		MYSQL_TYPE_BIT,
		MYSQL_TYPE_NEWDATE,
		MYSQL_TYPE_YEAR,
		MYSQL_TYPE_NULL,
		MYSQL_TYPE_ENUM,
		MYSQL_TYPE_SET,
		MYSQL_TYPE_TINY_BLOB,
		MYSQL_TYPE_MEDIUM_BLOB,
		MYSQL_TYPE_LONG_BLOB,
		MYSQL_TYPE_BLOB,
		MYSQL_TYPE_GEOMETRY : (* Unsupported MySQL-Data-Types *)
			sValue := CONCAT('CONVERT-ERROR: Unsupported MySQL-Data-Type: "', INT_TO_STRING(stQueryResult.astColumns[iCol-1].eType) );
			sValue := CONCAT(sValue, '"');
			MySql_GetStringValue := 16#80006008;
			;
	ELSE
		sValue := CONCAT('CONVERT-ERROR: Unknown MySQL-Data-Type: "', INT_TO_STRING(stQueryResult.astColumns[iCol-1].eType) );
		sValue := CONCAT(sValue, '"');
		MySql_GetStringValue := 16#80006007;
	END_CASE

END_IF

END_FUNCTION

// Device/Application/MYSQL/public/MySql_Version
FUNCTION MySql_Version : WORD
(*

 date     | release	| author  | Desc
----------+---------+------------------------------------------------------------
 21.03.14 |  3.8	| CM      | MySql_Query: New constant "gcMySql_tResponseCompliedlyReceived" 
 13.03.14 |  3.7	| CM      | MySql_Query: Initialisation of "stResultSet" now optional 
 02.07.12 |  3.6	| CM      | MySql_Query: BugFix for large SQL-Statements 
 17.04.12 |  3.5	| CM      | MySql_Query: BugFix for TIMEOUT error by "CALL <stored proc>"  
 25.01.12 |  3.4	| CM      | All: BugFix for large SQL statements 
 26.09.11 |  3.3	| CM      | MySql_Query: Clear complied result set before use 
 16.09.11 |  3.2	| CM      | MySql_Query: BugFix for large result sets 
 06.12.10 |  3.1    | CM      | MySql_GetStringValue: BugFix for Fieldtype 'TOD#'
 09.11.10 |  3.0    | CM      | MySql_Query: Optimize cycletime, "stResultSet" now VAR_IN_OUT prior VAR_OUTPUT  
 29.09.10 |  2.4    | CM      | MySql_Login: Bugfix for IP in dotted format
 28.09.10 |  2.3    | CM      | MySql_Login: Add DNS support for 750-881 and derivates
 28.09.10 |  2.2    | CM      | MySql_Login: Add error message when Login not allowed for this host
 19.08.10 |  2.1    | CM      | MySql_Query: ReceiveBuffer handling modified
 06.08.10 |  2.0	| CM      | Init - Switch from STRUCT "MySql" to FB "MySql_Context" 
 03.08.10 |  1.0	| CM      | Port to IEC 6-1131 
 22.06.09 |  0.0	| PEJ     | Original (C-Code)  
 
 *)
VAR_INPUT
END_VAR
VAR
	(* Current library version *)
	bMajor : BYTE := 16#03;
	bMinor : BYTE := 16#08;
END_VAR

MySql_Version := SHL(BYTE_TO_WORD(bMajor), 8) OR BYTE_TO_WORD(bMinor);

END_FUNCTION

// Device/Application/vis/Visualization
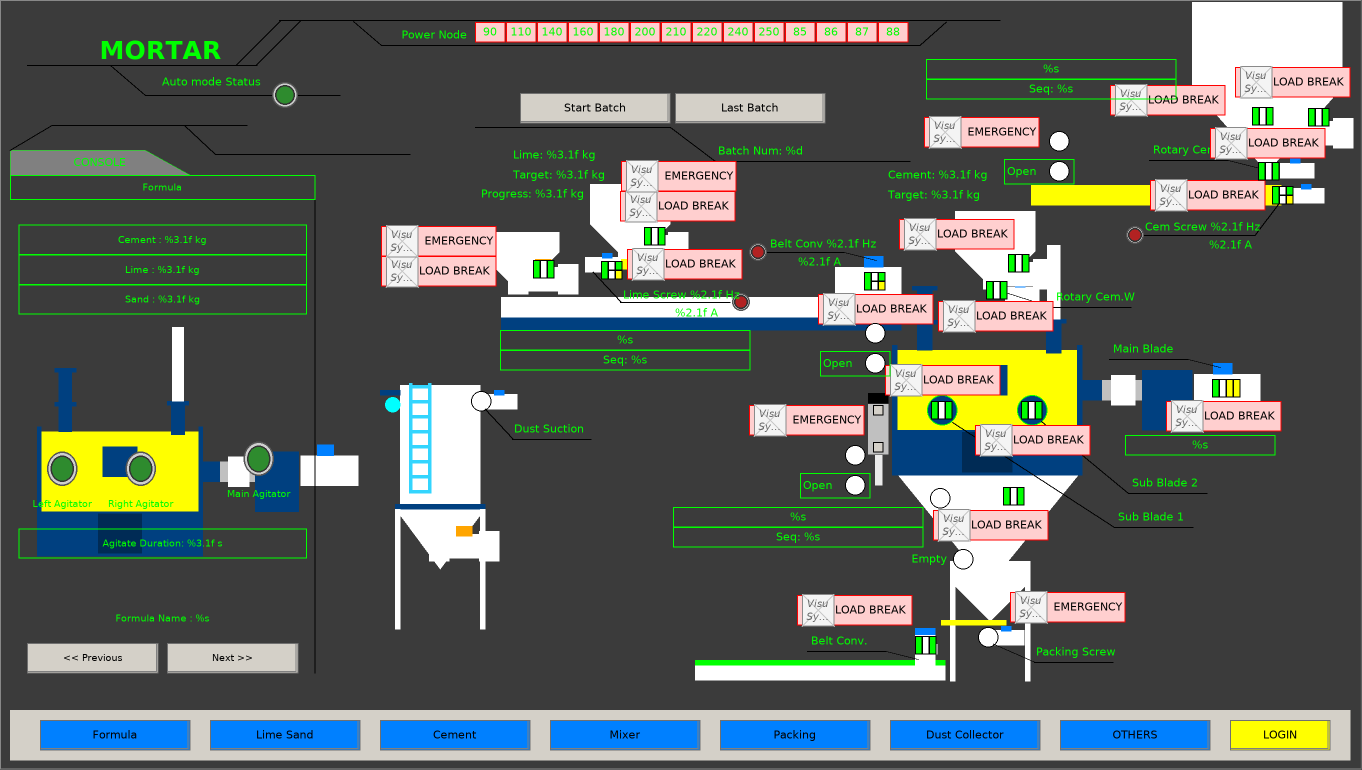
VISUALIZATION Visualization  // 1362x770
    Rectangle (800,473 70x25), "Open", colour toggle: DO381
    Rectangle (1004,159 70x25), "Open", colour toggle: DO371
    Line (1360,0) (1360,768)
    Rectangle (1031,185 250x20), angle 30
    Polygon (479,232) (559,232) (559,252) (519,292) (479,252)
    Rectangle (10,710 1340x50)
    Button (40,720 150x30), "Formula"
        OnMouseClick: FrameSelectionChange Selection=SelectedFrame=543ee2c1-9089-4e2a-a341-85b06829db8c, GlobSel=AssignType=Directly, SelType=Locally
    Button (210,720 150x30), "Lime Sand"
        OnMouseClick: FrameSelectionChange Selection=SelectedFrame=543ee2c1-9089-4e2a-a341-85b06829db8c, Selection=1, GlobSel=AssignType=Directly, SelType=Locally
    Button (380,720 150x30), "Cement"
        OnMouseClick: FrameSelectionChange Selection=SelectedFrame=543ee2c1-9089-4e2a-a341-85b06829db8c, Selection=2, GlobSel=AssignType=Directly, SelType=Locally
    Button (550,720 150x30), "Mixer"
        OnMouseClick: FrameSelectionChange Selection=SelectedFrame=543ee2c1-9089-4e2a-a341-85b06829db8c, Selection=3, GlobSel=AssignType=Directly, SelType=Locally
    Button (890,720 150x30), "Dust Collector"
        OnMouseClick: FrameSelectionChange Selection=SelectedFrame=543ee2c1-9089-4e2a-a341-85b06829db8c, Selection=4, GlobSel=AssignType=Directly, SelType=Locally
    Rectangle (1291,188 26x15), angle 30
    Rectangle (1301,184 10x5), angle 30
    Rectangle (1316,188 8x15), angle 30
    Line (1140,235) (1255,235)
    Line (1255,235) (1280,202)
    Polygon (1192,2) (1342,2) (1342,87) (1267,172) (1192,87)
    Rectangle (1280,163 26x15)
    Rectangle (1290,158 10x5)
    Rectangle (1306,163 8x15)
    Line (1149,160) (1228,160)
    Label (1150,140 100x20), "Rotary Cem"
    Line (1228,160) (1260,168)
    Group (1228,113 23x17)
        RoundedRectangle (0,5 20x30)
        RoundedRectangle (50,5 20x30)
        Rectangle (20,8 30x24)
        Rectangle (27,0 16x10)
    Group (1283,113 23x17)
        RoundedRectangle (0,5 20x30)
        RoundedRectangle (50,5 20x30)
        Rectangle (20,8 30x24)
        Rectangle (27,0 16x10)
    Group (1210,127 115x32), invisible if: DI183
        RoundedRectangle (0,1 115x30), "LOAD BREAK"
        Image (5,0 32x32), image: VisuSymbols.Symbols.Caution
    Polygon (955,211) (1035,211) (1035,251) (995,291) (955,251)
    Rectangle (885,165 120x20), "Cement: %3.1f kg", text variable: Cement_PRG.cement_weight
    Group (1005,282 20x15)
        Rectangle (0,5 26x15)
        Rectangle (10,0 10x5)
        Rectangle (26,5 8x15)
    Group (983,254 23x17)
        RoundedRectangle (0,5 20x30)
        RoundedRectangle (50,5 20x30)
        Rectangle (20,8 30x24)
        Rectangle (27,0 16x10)
    Rectangle (897,350 180x80)
    Polygon (973,567) (898,475) (1078,475) (1003,567) (988,567)
    Rectangle (967,365 40x30)
    Ellipse (1017,395 30x30)
    Ellipse (927,395 30x30)
    Rectangle (1046,323 15x30)
    Rectangle (1041,319 25x4)
    Rectangle (1077,345 5x130)
    Rectangle (892,345 5x130)
    Rectangle (897,430 180x45)
    Rectangle (962,432 50x40)
    Rectangle (1082,380 20x20)
    Rectangle (917,290 15x60)
    Rectangle (912,286 25x4)
    Rectangle (912,320 25x4)
    Rectangle (1102,380 40x20)
    Rectangle (1142,370 50x60)
    Rectangle (1111,375 24x30)
    Rectangle (1194,374 51x30)
    Rectangle (1213,363 19x11)
    Rectangle (1245,374 15x30)
    Rectangle (968,510 40x30)
    Rectangle (868,404 20x50)
    Rectangle (875,455 7x30)
    Line (1041,421) (1128,493)
    Line (1128,493) (1207,493)
    Label (1129,473 100x20), "Sub Blade 2"
    Line (952,422) (1114,527)
    Line (1114,527) (1193,527)
    Label (1115,507 100x20), "Sub Blade 1"
    Line (1109,359) (1188,359)
    Label (1110,339 100x20), "Main Blade"
    Line (1188,359) (1220,367)
    RoundedRectangle (1047,245 13x74)
    Group (976,490 23x17)
        RoundedRectangle (0,5 20x30)
        RoundedRectangle (50,5 20x30)
        Rectangle (20,8 30x24)
        Rectangle (27,0 16x10)
    Group (508,259 23x17)
        RoundedRectangle (0,5 20x30)
        RoundedRectangle (50,5 20x30)
        Rectangle (20,8 30x24)
        Rectangle (27,0 16x10)
    Rectangle (501,315 400x15), angle 330
    Rectangle (501,297 400x20), angle 330
    Rectangle (850,267 51x30)
    Rectangle (864,256 19x11)
    Rectangle (835,267 15x30)
    Line (765,252) (844,252)
    Line (844,252) (876,260)
    Polygon (590,184) (670,184) (670,224) (630,264) (590,224)
    Rectangle (510,145 120x20), "Lime: %3.1f kg", text variable: LimeSand.lime_weight
    Group (618,227 23x17)
        RoundedRectangle (0,5 20x30)
        RoundedRectangle (50,5 20x30)
        Rectangle (20,8 30x24)
        Rectangle (27,0 16x10)
    Rectangle (621,259 100x10), angle 30
    Line (1052,307) (1131,307)
    Label (1053,287 100x20), "Rotary Cem.W"
    Line (1005,292) (1052,307)
    Rectangle (868,393 20x10)
    Ellipse (845,445 20x20), colour toggle: DI224
    Ellipse (845,475 20x20), colour toggle: DI225
    Label (898,549 52x20), "Empty"
    Rectangle (950,581 5x100)
    Rectangle (1025,581 5x100)
    Polygon (950,561) (1030,561) (1030,581) (990,621) (950,581)
    Ellipse (953,549 20x20), colour toggle: DI264
    Rectangle (941,620 65x5), angle 30
    Rectangle (991,630 26x15), angle 30
    Rectangle (1001,626 10x5), angle 30
    Rectangle (1016,630 8x15), angle 30
    Ellipse (978,627 20x20)
    Label (1033,642 100x20), "Packing Screw"
    Line (1034,662) (1113,662)
    Line (1034,662) (993,644)
    Rectangle (695,665 250x15)
    Rectangle (915,628 20x7)
    Rectangle (695,660 250x5)
    Rectangle (915,635 20x30)
    Rectangle (932,644 5x10)
    Line (807,651) (886,651)
    Label (808,631 100x20), "Belt Conv."
    Line (886,651) (918,659)
    Group (380,383 231x246)
        Rectangle (20,2 80x120)
        Rectangle (104,11 26x15), angle 30
        Rectangle (114,7 10x5), angle 30
        Rectangle (129,11 8x15), angle 30
        Ellipse (91,8 20x20)
        Label (131,36 100x20), "Dust Suction"
        Line (132,56) (211,56)
        Line (133,56) (105,26)
        Rectangle (0,7 20x5)
        Ellipse (5,14 15x15)
        Rectangle (29,0 3x110)
        Rectangle (48,0 3x110)
        Rectangle (30,107 20x3)
        Rectangle (30,92 20x3)
        Rectangle (30,77 20x3)
        Rectangle (30,62 20x3)
        Rectangle (30,47 20x3)
        Rectangle (30,32 20x3)
        Rectangle (30,17 20x3)
        Rectangle (30,2 20x3)
        Polygon (20,126) (100,126) (100,132) (60,186) (20,132)
        Group (49,143 23x17)
            RoundedRectangle (0,5 20x30)
            RoundedRectangle (50,5 20x30)
            Rectangle (20,8 30x24)
            Rectangle (27,0 16x10)
        Rectangle (15,121 90x5)
        Rectangle (15,126 5x120)
        Rectangle (100,126 5x120)
    Button (1060,720 150x30), "OTHERS"
        OnMouseClick: FrameSelectionChange Selection=SelectedFrame=543ee2c1-9089-4e2a-a341-85b06829db8c, Selection=5, GlobSel=AssignType=Directly, SelType=Locally
    Button (1230,720 100x30), "LOGIN"
    Group (818,293 115x32), invisible if: DI191
        RoundedRectangle (0,1 115x30), "LOAD BREAK"
        Image (5,0 32x32), image: VisuSymbols.Symbols.Caution
    Group (938,300 115x32), invisible if: DI184
        RoundedRectangle (0,1 115x30), "LOAD BREAK"
        Image (5,0 32x32), image: VisuSymbols.Symbols.Caution
    Group (885,364 115x32), invisible if: DI207
        RoundedRectangle (0,1 115x30), "LOAD BREAK"
        Image (5,0 32x32), image: VisuSymbols.Symbols.Caution
    Group (975,424 115x32), invisible if: DI208
        RoundedRectangle (0,1 115x30), "LOAD BREAK"
        Image (5,0 32x32), image: VisuSymbols.Symbols.Caution
    Group (1166,400 115x32), invisible if: DI238
        RoundedRectangle (0,1 115x30), "LOAD BREAK"
        Image (5,0 32x32), image: VisuSymbols.Symbols.Caution
    Group (1150,179 115x32), invisible if: DI185
        RoundedRectangle (0,1 115x30), "LOAD BREAK"
        Image (5,0 32x32), image: VisuSymbols.Symbols.Caution
    Group (627,248 115x32), invisible if: DI192
        RoundedRectangle (0,1 115x30), "LOAD BREAK"
        Image (5,0 32x32), image: VisuSymbols.Symbols.Caution
    Rectangle (592,257 26x15), angle 30
    Rectangle (602,253 10x5), angle 30
    Rectangle (585,257 8x15), angle 30
    Line (620,302) (730,302)
    Line (621,302) (593,272)
    Rectangle (10,175 350x500)
    Polygon (10,150) (80,150) (145,150) (190,175) (10,175), "CONSOLE"
    Frame (10,175 350x500)
        shows formula()
        shows lime()
        shows cement()
        shows mixer()
        shows dust()
        shows other()
        shows packing()
        shows login()
    Line (27,65) (257,65)
    Line (279,20) (1000,20)
    Line (256,65) (301,20)
    Line (236,65) (281,20)
    Label (0,35 321x30), "MORTAR"
    Group (620,190 115x32), invisible if: DI193
        RoundedRectangle (0,1 115x30), "LOAD BREAK"
        Image (5,0 32x32), image: VisuSymbols.Symbols.Caution
    Group (381,255 115x32), invisible if: DI195
        RoundedRectangle (0,1 115x30), "LOAD BREAK"
        Image (5,0 32x32), image: VisuSymbols.Symbols.Caution
    Group (899,218 115x32), invisible if: DI186
        RoundedRectangle (0,1 115x30), "LOAD BREAK"
        Image (5,0 32x32), image: VisuSymbols.Symbols.Caution
    Group (1235,66 115x32), invisible if: DI182
        RoundedRectangle (0,1 115x30), "LOAD BREAK"
        Image (5,0 32x32), image: VisuSymbols.Symbols.Caution
    Group (1110,84 115x32), invisible if: DI181
        RoundedRectangle (0,1 115x30), "LOAD BREAK"
        Image (5,0 32x32), image: VisuSymbols.Symbols.Caution
    Rectangle (601,261 7x18), colour toggle: DI132
    Rectangle (608,261 7x9), colour toggle: DO322
    Rectangle (615,261 7x9), colour toggle: DI152
    Rectangle (533,260 7x18), colour toggle: DI135
    Rectangle (540,260 7x18), colour toggle: DO325
    Rectangle (547,260 7x18), colour toggle: DI155
    Rectangle (644,227 7x18), colour toggle: DI133
    Rectangle (651,227 7x18), colour toggle: DO323
    Rectangle (658,227 7x18), colour toggle: DI153
    Rectangle (864,272 7x18), colour toggle: DI131
    Rectangle (871,272 7x9), colour toggle: DO321
    Rectangle (878,272 7x9), colour toggle: DI151
    Rectangle (1008,254 7x18), colour toggle: DI126
    Rectangle (1015,254 7x18), colour toggle: DO316
    Rectangle (1022,254 7x18), colour toggle: DI146
    Rectangle (986,281 7x18), colour toggle: DI124
    Rectangle (993,281 7x18), colour toggle: DO314
    Rectangle (1000,281 7x18), colour toggle: DI144
    Rectangle (1272,186 7x18), colour toggle: DI125
    Rectangle (1279,186 7x9), colour toggle: DO315
    Rectangle (1286,186 7x9), colour toggle: DI145
    Rectangle (1258,162 7x18), colour toggle: DI123
    Rectangle (1265,162 7x18), colour toggle: DO313
    Rectangle (1272,162 7x18), colour toggle: DI143
    Rectangle (1308,108 7x18), colour toggle: DI122
    Rectangle (1315,108 7x18), colour toggle: DO312
    Rectangle (1322,108 7x18), colour toggle: DI142
    Rectangle (1252,107 7x18), colour toggle: DI121
    Rectangle (1259,107 7x18), colour toggle: DO311
    Rectangle (1266,107 7x18), colour toggle: DI141
    Button (720,720 150x30), "Packing"
        OnMouseClick: FrameSelectionChange Selection=SelectedFrame=543ee2c1-9089-4e2a-a341-85b06829db8c, Selection=6, GlobSel=AssignType=Directly, SelType=Locally
    Line (110,65) (145,95)
    Line (145,95) (340,95)
    Label (159,67 150x30), "Auto mode Status"
    Line (52,125) (247,125)
    Line (215,154) (410,154)
    Line (10,150) (52,125)
    Line (184,125) (215,154)
    Button (520,93 150x30), "Start Batch", invisible if: Automode.show_start
        tap Automode.run_batch
    Button (675,93 150x30), "Last Batch"
        tap Automode.last_batch
    Line (475,127) (670,127)
    Line (715,161) (910,161)
    Line (670,127) (715,161)
    Rectangle (715,136 200x30), "Batch Num: %d"
    Lamp1 (270,80 30x30), variable: Automode.auto_mode, style: Lamp-Lamp1-Green
    Rectangle (510,165 120x20), "Target: %3.1f kg", text variable: LimeSand.lime_targetfix
    Rectangle (885,185 120x20), "Target: %3.1f kg", text variable: Cement_PRG.cement_targetfix
    Rectangle (1212,379 7x18), colour toggle: DI173
    Rectangle (1219,379 7x18), colour toggle: DO347
    Rectangle (1226,379 7x18), colour toggle: DI254
    Rectangle (1233,379 7x18), colour toggle: DI256
    Rectangle (1021,401 7x18), colour toggle: DI172
    Rectangle (1028,401 7x18), colour toggle: DO346
    Rectangle (1035,401 7x18), colour toggle: DI258
    Rectangle (931,401 7x18), colour toggle: DI171
    Rectangle (938,401 7x18), colour toggle: DO345
    Rectangle (945,401 7x18), colour toggle: DI257
    Rectangle (1003,487 7x18), colour toggle: DI127
    Rectangle (1010,487 7x18), colour toggle: DO317
    Rectangle (1017,487 7x18), colour toggle: DI147
    Rectangle (915,636 7x18), colour toggle: DI128
    Rectangle (922,636 7x18), colour toggle: DO318
    Rectangle (929,636 7x18), colour toggle: DI148
    Rectangle (608,270 7x9), colour toggle: DO335
    Rectangle (615,270 7x9), colour toggle: DI165
    Lamp1 (731,292 20x20), variable: DI166, style: Lamp-Lamp1-Red
    Lamp1 (748,242 20x20), variable: DI164, style: Lamp-Lamp1-Red
    Lamp1 (1125,225 20x20), variable: DI162, style: Lamp-Lamp1-Red
    Rectangle (620,280 150x30), "Lime Screw %2.1f Hz", text variable: LimeSand.screw_Hz
    Rectangle (767,229 150x30), "Belt Conv %2.1f Hz", text variable: LimeSand.belt_Hz
    Rectangle (1142,212 150x30), "Cem Screw %2.1f Hz", text variable: Cement_PRG.screw_Hz
    Rectangle (871,281 7x9), colour toggle: DO333
    Rectangle (878,281 7x9), colour toggle: DI163
    Rectangle (1286,195 7x9), colour toggle: DI161
    Rectangle (1279,195 7x9), colour toggle: DO331
    Group (933,509 115x32), invisible if: DI187
        RoundedRectangle (0,1 115x30), "LOAD BREAK"
        Image (5,0 32x32), image: VisuSymbols.Symbols.Caution
    Group (797,594 115x32), invisible if: DI188
        RoundedRectangle (0,1 115x30), "LOAD BREAK"
        Image (5,0 32x32), image: VisuSymbols.Symbols.Caution
    Ellipse (1049,131 20x20), colour toggle: DI204
    Ellipse (1049,161 20x20), colour toggle: DI203
    Rectangle (873,405 10x10), colour toggle: DI222
    Rectangle (873,442 10x10), colour toggle: DI223
    Rectangle (475,22 30x20), "90", colour toggle: DI136
    Rectangle (506,22 30x20), "110", colour toggle: DI137
    Rectangle (537,22 30x20), "140", colour toggle: DI156
    Rectangle (568,22 30x20), "160", colour toggle: DI178
    Rectangle (599,22 30x20), "180", colour toggle: DI196
    Rectangle (630,22 30x20), "200", colour toggle: DI201
    Rectangle (661,22 30x20), "210", colour toggle: DI211
    Rectangle (785,22 30x20), "85", colour toggle: DI217
    Rectangle (816,22 30x20), "86", colour toggle: DI218
    Rectangle (692,22 30x20), "220", colour toggle: DI221
    Rectangle (723,22 30x20), "240", colour toggle: DI241
    Rectangle (754,22 30x20), "250", colour toggle: DI251
    Line (381,45) (920,45)
    Line (353,21) (381,45)
    Label (370,25 100x20), "Power Node"
    Rectangle (500,330 250x20), "%s", text variable: LimeSand.lime_alarm
    Rectangle (926,59 250x20), "%s", text variable: Cement_PRG.cement_alarm
    Rectangle (847,22 30x20), "87", colour toggle: DI247
    Rectangle (878,22 30x20), "88", colour toggle: DI248
    Line (946,22) (920,45)
    Group (924,116 115x32), invisible if: DI205
        RoundedRectangle (0,1 115x30), "EMERGENCY"
        Image (5,0 32x32), image: VisuSymbols.Symbols.Caution
    Group (621,160 115x32), invisible if: DI214
        RoundedRectangle (0,1 115x30), "EMERGENCY"
        Image (5,0 32x32), image: VisuSymbols.Symbols.Caution
    Group (381,225 115x32), invisible if: DI214
        RoundedRectangle (0,1 115x30), "EMERGENCY"
        Image (5,0 32x32), image: VisuSymbols.Symbols.Caution
    Group (749,404 115x32), invisible if: DI233
        RoundedRectangle (0,1 115x30), "EMERGENCY"
        Image (5,0 32x32), image: VisuSymbols.Symbols.Caution
    Rectangle (673,507 250x20), "%s", text variable: Mixer_PRG.mixer_alarm
    Ellipse (865,323 20x20), colour toggle: DI226
    Rectangle (820,351 70x25), "Open", colour toggle: DO326
    Ellipse (865,353 20x20), colour toggle: DI227
    Rectangle (478,184 120x20), "Progress: %3.1f kg", text variable: LimeSand.lime_progress
    Ellipse (930,488 20x20), colour toggle: DI265
    Rectangle (621,303 100x20), "%2.1f A", text variable: LimeSand.lime_amp
    Rectangle (744,252 100x20), "%2.1f A", text variable: LimeSand.belt_amp
    Rectangle (1155,235 100x20), "%2.1f A", text variable: Cement_PRG.cement_amp
    Rectangle (500,350 250x20), "Seq: %s", text variable: LimeSand.lime_seq
    Rectangle (673,527 250x20), "Seq: %s", text variable: Mixer_PRG.mixer_seq
    Rectangle (926,79 250x20), "Seq: %s", text variable: Cement_PRG.cement_seq
    RoundedRectangle (1010,592 115x30), "EMERGENCY"
    Image (1015,591 32x32), image: VisuSymbols.Symbols.Caution
    Rectangle (1125,435 150x20), "%s", text variable: Mixer_PRG.tmp_agitate
END_VISUALIZATION

// Device/Application/vis/formula
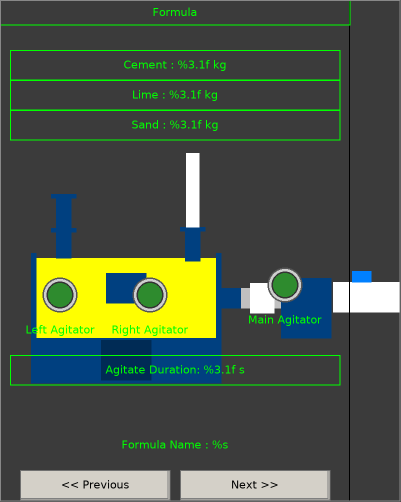
VISUALIZATION formula  // 401x502
    Group (31,153 279x179)
        Rectangle (5,105 180x80)
        Rectangle (75,120 40x30)
        Rectangle (154,78 15x30)
        Rectangle (149,74 25x4)
        Rectangle (185,100 5x130)
        Rectangle (0,100 5x130)
        Rectangle (5,185 180x45)
        Rectangle (70,187 50x40)
        Rectangle (190,135 20x20)
        Rectangle (25,45 15x60)
        Rectangle (20,41 25x4)
        Rectangle (20,75 25x4)
        Rectangle (210,135 40x20)
        Rectangle (250,125 50x60)
        Rectangle (219,130 24x30)
        Rectangle (302,129 51x30)
        Rectangle (321,118 19x11)
        Rectangle (353,129 15x30)
        RoundedRectangle (155,0 13x74)
    Line (349,0) (349,500)
    Rectangle (0,0 350x25), "Formula"
    Button (20,470 150x30), "<< Previous"
        tap Formula.prev_formula
    Button (180,470 150x30), "Next >>"
        tap Formula.next_formula
    Rectangle (10,50 330x30), "Cement : %3.1f kg", text variable: Formula.cement_target
    Rectangle (10,80 330x30), "Lime : %3.1f kg", text variable: Formula.lime_target
    Rectangle (10,110 330x30), "Sand : %3.1f kg", text variable: Formula.sand_target
    Rectangle (10,430 330x30), "Formula Name : %s", text variable: Formula.formula_name
    Lamp1 (130,275 40x40), variable: Formula.Formula_Loader_0.right_agitate, style: Lamp-Lamp1-Green
    Lamp1 (40,275 40x40), variable: Formula.Formula_Loader_0.left_agitate, style: Lamp-Lamp1-Green
    Lamp1 (265,265 40x40), variable: Formula.Formula_Loader_0.main_agitate, style: Lamp-Lamp1-Green
    Label (10,320 100x20), "Left Agitator"
    Label (100,320 100x20), "Right Agitator"
    Label (235,310 100x20), "Main Agitator"
    Rectangle (10,355 330x30), "Agitate Duration: %3.1f s", text variable: Formula.Formula_Loader_0.agitate_time
END_VISUALIZATION

// Device/Application/vis/packing
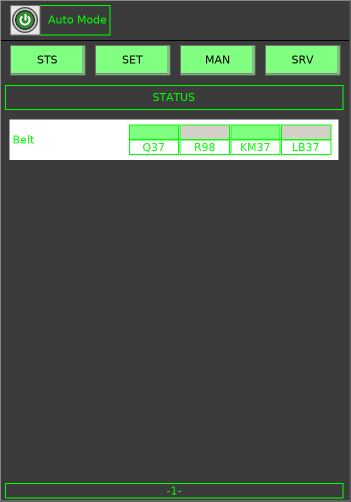
VISUALIZATION packing  // 351x502
    Line (349,0) (349,500)
    Line (349,0) (349,500)
    Frame (5,85 340x415)
        shows packing_0()
        shows packing_1()
        shows packing_2()
        shows packing_3()
    Button (10,45 75x30), "STS"
        OnMouseClick: FrameSelectionChange Selection=SelectedFrame=38382966-a585-44b7-b9fb-7a78fd5e578f, GlobSel=AssignType=Directly, SelType=Locally
    Button (95,45 75x30), "SET"
        OnMouseClick: FrameSelectionChange Selection=SelectedFrame=38382966-a585-44b7-b9fb-7a78fd5e578f, Selection=1, GlobSel=AssignType=Directly, SelType=Locally
    Button (180,45 75x30), "MAN"
        OnMouseClick: FrameSelectionChange Selection=SelectedFrame=38382966-a585-44b7-b9fb-7a78fd5e578f, Selection=2, GlobSel=AssignType=Directly, SelType=Locally
    Button (265,45 75x30), "SRV"
        OnMouseClick: FrameSelectionChange Selection=SelectedFrame=38382966-a585-44b7-b9fb-7a78fd5e578f, Selection=3, GlobSel=AssignType=Directly, SelType=Locally
    Line (0,40) (349,40)
    Rectangle (10,5 100x30), "Auto Mode"
    PowerSwitch (10,5 30x30), variable: Automode.auto_packing, behaviour: TOGGLE, style: Switch-PowerSwitch-Green
END_VISUALIZATION

// Device/Application/vis/lime
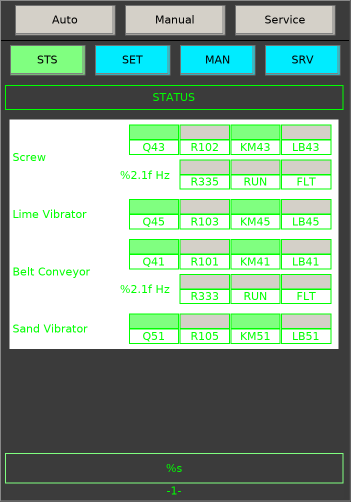
VISUALIZATION lime  // 351x502
    Line (349,0) (349,500)
    Button (15,5 100x30), "Auto", colour toggle: LimeSand.auto_lime
        tap LimeSand.auto_limex
        OnMouseClick: FrameSelectionChange Selection=SelectedFrame=f95ddd8c-2b3d-468a-8364-643e41e106f5, GlobSel=AssignType=Directly, SelType=Locally
    Button (125,5 100x30), "Manual", colour toggle: LimeSand.manual_lime
        tap LimeSand.manual_limex
        OnMouseClick: FrameSelectionChange Selection=SelectedFrame=f95ddd8c-2b3d-468a-8364-643e41e106f5, Selection=2, GlobSel=AssignType=Directly, SelType=Locally
    Button (235,5 100x30), "Service", colour toggle: LimeSand.service_lime
        tap LimeSand.service_limex
        OnMouseClick: FrameSelectionChange Selection=SelectedFrame=f95ddd8c-2b3d-468a-8364-643e41e106f5, Selection=3, GlobSel=AssignType=Directly, SelType=Locally
    Button (10,45 75x30), "STS"
        OnMouseClick: FrameSelectionChange Selection=SelectedFrame=f95ddd8c-2b3d-468a-8364-643e41e106f5, GlobSel=AssignType=Directly, SelType=Locally
    Frame (5,85 340x415)
        shows lime_0()
        shows lime_1()
        shows lime_2()
        shows lime_3()
    Button (95,45 75x30), "SET", colour toggle: LimeSand.auto_lime
        OnMouseClick: FrameSelectionChange Selection=SelectedFrame=f95ddd8c-2b3d-468a-8364-643e41e106f5, Selection=1, GlobSel=AssignType=Directly, SelType=Locally
    Button (180,45 75x30), "MAN", colour toggle: LimeSand.manual_lime
        OnMouseClick: FrameSelectionChange Selection=SelectedFrame=f95ddd8c-2b3d-468a-8364-643e41e106f5, Selection=2, GlobSel=AssignType=Directly, SelType=Locally
    Button (265,45 75x30), "SRV", colour toggle: LimeSand.service_lime
        OnMouseClick: FrameSelectionChange Selection=SelectedFrame=f95ddd8c-2b3d-468a-8364-643e41e106f5, Selection=3, GlobSel=AssignType=Directly, SelType=Locally
    Line (0,40) (349,40)
END_VISUALIZATION

// Device/Application/vis/cement
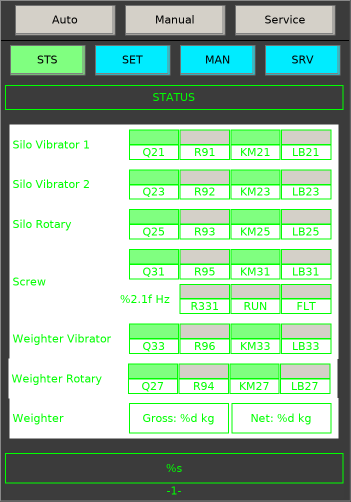
VISUALIZATION cement  // 351x502
    Line (349,0) (349,500)
    Button (15,5 100x30), "Auto", colour toggle: Cement_PRG.auto_cement
        tap Cement_PRG.auto_cementx
        OnMouseClick: FrameSelectionChange Selection=SelectedFrame=f95ddd8c-2b3d-468a-8364-643e41e106f5, GlobSel=AssignType=Directly, SelType=Locally
    Button (125,5 100x30), "Manual", colour toggle: Cement_PRG.manual_cement
        tap Cement_PRG.manual_cementx
        OnMouseClick: FrameSelectionChange Selection=SelectedFrame=f95ddd8c-2b3d-468a-8364-643e41e106f5, Selection=2, GlobSel=AssignType=Directly, SelType=Locally
    Button (235,5 100x30), "Service", colour toggle: Cement_PRG.service_cement
        tap Cement_PRG.service_cementx
        OnMouseClick: FrameSelectionChange Selection=SelectedFrame=f95ddd8c-2b3d-468a-8364-643e41e106f5, Selection=3, GlobSel=AssignType=Directly, SelType=Locally
    Button (10,45 75x30), "STS"
        OnMouseClick: FrameSelectionChange Selection=SelectedFrame=f95ddd8c-2b3d-468a-8364-643e41e106f5, GlobSel=AssignType=Directly, SelType=Locally
    Frame (5,85 340x415)
        shows cement_0()
        shows cement_1()
        shows cement_2()
        shows cement_3()
    Button (95,45 75x30), "SET", colour toggle: Cement_PRG.auto_cement
        OnMouseClick: FrameSelectionChange Selection=SelectedFrame=f95ddd8c-2b3d-468a-8364-643e41e106f5, Selection=1, GlobSel=AssignType=Directly, SelType=Locally
    Button (180,45 75x30), "MAN", colour toggle: Cement_PRG.manual_cement
        OnMouseClick: FrameSelectionChange Selection=SelectedFrame=f95ddd8c-2b3d-468a-8364-643e41e106f5, Selection=2, GlobSel=AssignType=Directly, SelType=Locally
    Button (265,45 75x30), "SRV", colour toggle: Cement_PRG.service_cement
        OnMouseClick: FrameSelectionChange Selection=SelectedFrame=f95ddd8c-2b3d-468a-8364-643e41e106f5, Selection=3, GlobSel=AssignType=Directly, SelType=Locally
    Line (0,40) (349,40)
END_VISUALIZATION

// Device/Application/vis/mixer
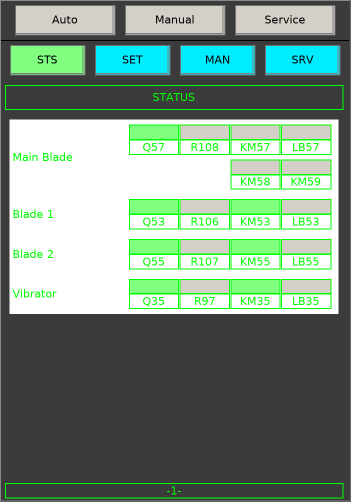
VISUALIZATION mixer  // 351x502
    Line (349,0) (349,500)
    Button (15,5 100x30), "Auto", colour toggle: Mixer_PRG.auto_mixer
        tap Mixer_PRG.auto_mixerx
        OnMouseClick: FrameSelectionChange Selection=SelectedFrame=13b2a05a-9515-4b6b-aaa5-d4f3704da2e4, GlobSel=AssignType=Directly, SelType=Locally
    Button (125,5 100x30), "Manual", colour toggle: Mixer_PRG.manual_mixer
        tap Mixer_PRG.manual_mixerx
        OnMouseClick: FrameSelectionChange Selection=SelectedFrame=13b2a05a-9515-4b6b-aaa5-d4f3704da2e4, Selection=2, GlobSel=AssignType=Directly, SelType=Locally
    Button (235,5 100x30), "Service", colour toggle: Mixer_PRG.service_mixer
        tap Mixer_PRG.service_mixerx
        OnMouseClick: FrameSelectionChange Selection=SelectedFrame=13b2a05a-9515-4b6b-aaa5-d4f3704da2e4, Selection=3, GlobSel=AssignType=Directly, SelType=Locally
    Frame (5,85 340x415)
        shows mixer_0()
        shows mixer_1()
        shows mixer_2()
        shows mixer_3()
    Button (10,45 75x30), "STS"
        OnMouseClick: FrameSelectionChange Selection=SelectedFrame=13b2a05a-9515-4b6b-aaa5-d4f3704da2e4, GlobSel=AssignType=Directly, SelType=Locally
    Button (95,45 75x30), "SET", colour toggle: Mixer_PRG.auto_mixer
        OnMouseClick: FrameSelectionChange Selection=SelectedFrame=13b2a05a-9515-4b6b-aaa5-d4f3704da2e4, Selection=1, GlobSel=AssignType=Directly, SelType=Locally
    Button (180,45 75x30), "MAN", colour toggle: Mixer_PRG.manual_mixer
        OnMouseClick: FrameSelectionChange Selection=SelectedFrame=13b2a05a-9515-4b6b-aaa5-d4f3704da2e4, Selection=2, GlobSel=AssignType=Directly, SelType=Locally
    Button (265,45 75x30), "SRV", colour toggle: Mixer_PRG.service_mixer
        OnMouseClick: FrameSelectionChange Selection=SelectedFrame=13b2a05a-9515-4b6b-aaa5-d4f3704da2e4, Selection=3, GlobSel=AssignType=Directly, SelType=Locally
    Line (0,40) (349,40)
END_VISUALIZATION

// Device/Application/vis/dust
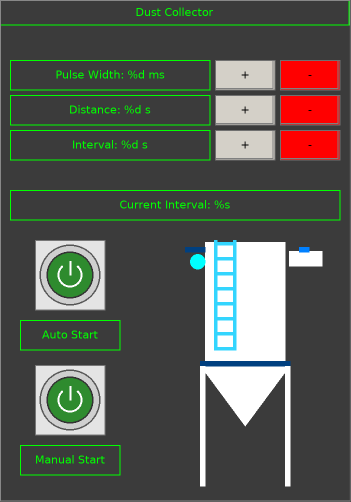
VISUALIZATION dust  // 351x502
    Line (349,0) (349,500)
    Rectangle (0,0 349x25), "Dust Collector"
    Rectangle (10,60 200x30), "Pulse Width: %d ms", text variable: Automode.pulse
    Rectangle (10,95 200x30), "Distance: %d s", text variable: Automode.distance
    Rectangle (10,130 200x30), "Interval: %d s", text variable: Automode.interval
    Rectangle (10,190 330x30), "Current Interval: %s", text variable: Automode.DC_0.tmp_int
    Button (215,60 60x30), "+"
        tap Automode.add_pulse
    Button (280,60 60x30), "-"
        tap Automode.sub_pulse
    Button (215,95 60x30), "+"
        tap Automode.add_distance
    Button (280,95 60x30), "-"
        tap Automode.sub_distance
    Button (215,130 60x30), "+"
        tap Automode.add_interval
    Button (280,130 60x30), "-"
        tap Automode.sub_interval
    PowerSwitch (35,365 70x70), variable: Automode.manual_dust, behaviour: TOGGLE, style: Switch-PowerSwitch-Green
    PowerSwitch (35,240 70x70), variable: Automode.auto_dust, behaviour: TOGGLE, style: Switch-PowerSwitch-Green
    Rectangle (20,320 100x30), "Auto Start"
    Rectangle (20,445 100x30), "Manual Start"
    Group (185,240 137x246)
        Rectangle (20,2 80x120)
        Rectangle (104,11 26x15), angle 30
        Rectangle (114,7 10x5), angle 30
        Rectangle (129,11 8x15), angle 30
        Rectangle (0,7 20x5)
        Ellipse (5,14 15x15)
        Rectangle (29,0 3x110)
        Rectangle (48,0 3x110)
        Rectangle (30,107 20x3)
        Rectangle (30,92 20x3)
        Rectangle (30,77 20x3)
        Rectangle (30,62 20x3)
        Rectangle (30,47 20x3)
        Rectangle (30,32 20x3)
        Rectangle (30,17 20x3)
        Rectangle (30,2 20x3)
        Polygon (20,126) (100,126) (100,132) (60,186) (20,132)
        Rectangle (15,121 90x5)
        Rectangle (15,126 5x120)
        Rectangle (100,126 5x120)
END_VISUALIZATION

// Device/Application/vis/other
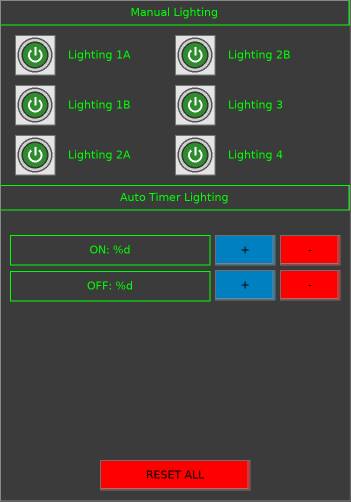
VISUALIZATION other  // 351x502
    Line (349,0) (349,500)
    PowerSwitch (15,35 40x40), variable: PLC_PRG.lighting1A, behaviour: TOGGLE, style: Switch-PowerSwitch-Green
    PowerSwitch (15,85 40x40), variable: PLC_PRG.lighting1B, behaviour: TOGGLE, style: Switch-PowerSwitch-Green
    PowerSwitch (15,135 40x40), variable: PLC_PRG.lighting2A, behaviour: TOGGLE, style: Switch-PowerSwitch-Green
    PowerSwitch (175,35 40x40), variable: PLC_PRG.lighting2B, behaviour: TOGGLE, style: Switch-PowerSwitch-Green
    PowerSwitch (175,85 40x40), variable: PLC_PRG.lighting3, behaviour: TOGGLE, style: Switch-PowerSwitch-Green
    PowerSwitch (175,135 40x40), variable: PLC_PRG.lighting4, behaviour: TOGGLE, style: Switch-PowerSwitch-Green
    Label (65,40 100x30), "Lighting 1A"
    Label (65,90 100x30), "Lighting 1B"
    Label (225,40 100x30), "Lighting 2B"
    Label (65,140 100x30), "Lighting 2A"
    Label (225,140 100x30), "Lighting 4"
    Label (225,90 100x30), "Lighting 3"
    Rectangle (0,0 349x25), "Manual Lighting"
    Rectangle (0,185 349x25), "Auto Timer Lighting"
    Rectangle (10,235 200x30), "ON: %d", text variable: Formula.jamnyala
    Rectangle (10,271 200x30), "OFF: %d", text variable: Formula.jammati
    Button (215,235 60x30), "+"
        tap Formula.tomboltambah
    Button (280,235 60x30), "-"
        tap Formula.tombolkurang
    Button (215,270 60x30), "+"
        tap Formula.tomboltambahmati
    Button (280,270 60x30), "-"
        tap Formula.tombolkurangmati
    Button (100,460 150x30), "RESET ALL"
        tap Automode.reset_all
END_VISUALIZATION

// Device/Application/vis/cement_1
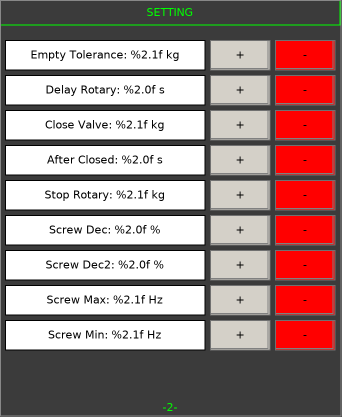
VISUALIZATION cement_1  // 342x417
    Rectangle (0,0 340x25), "SETTING"
    RoundedRectangle (5,40 200x30), "Empty Tolerance: %2.1f kg", text variable: Cement_PRG.cement_tolerance
    Button (210,40 60x30), "+"
        tap Cement_PRG.add_tolerance
    Button (275,40 60x30), "-"
        tap Cement_PRG.sub_tolerance
    RoundedRectangle (5,75 200x30), "Delay Rotary: %2.0f s", text variable: Cement_PRG.delay_rotary
    Button (210,75 60x30), "+"
        tap Cement_PRG.add_delayrotary
    Button (275,75 60x30), "-"
        tap Cement_PRG.sub_delayrotary
    RoundedRectangle (5,110 200x30), "Close Valve: %2.1f kg", text variable: Cement_PRG.closevalve_value
    Button (210,110 60x30), "+"
        tap Cement_PRG.add_close
    Button (275,110 60x30), "-"
        tap Cement_PRG.sub_close
    RoundedRectangle (5,145 200x30), "After Closed: %2.0f s", text variable: Cement_PRG.afterclose
    Button (210,145 60x30), "+"
        tap Cement_PRG.add_afterclose
    Button (275,145 60x30), "-"
        tap Cement_PRG.sub_afterclose
    RoundedRectangle (5,180 200x30), "Stop Rotary: %2.1f kg", text variable: Cement_PRG.stoprot
    Button (210,180 60x30), "+"
        tap Cement_PRG.add_stoprot
    Button (275,180 60x30), "-"
        tap Cement_PRG.sub_stoprot
    RoundedRectangle (5,215 200x30), "Screw Dec: %2.0f %", text variable: Cement_PRG.slow_screw
    Button (210,215 60x30), "+"
        tap Cement_PRG.add_slowscrew
    Button (275,215 60x30), "-"
        tap Cement_PRG.sub_slowscrew
    RoundedRectangle (5,285 200x30), "Screw Max: %2.1f Hz", text variable: Cement_PRG.max_screw
    Button (210,285 60x30), "+"
        tap Cement_PRG.add_maxscrew
    Button (275,285 60x30), "-"
        tap Cement_PRG.sub_maxscrew
    RoundedRectangle (5,320 200x30), "Screw Min: %2.1f Hz", text variable: Cement_PRG.min_screw
    Button (210,320 60x30), "+"
        tap Cement_PRG.add_minscrew
    Button (275,320 60x30), "-"
        tap Cement_PRG.sub_minscrew
    RoundedRectangle (5,250 200x30), "Screw Dec2: %2.0f %", text variable: Cement_PRG.slow_screw2
    Button (210,250 60x30), "+"
        tap Cement_PRG.add_slowscrew2
    Button (275,250 60x30), "-"
        tap Cement_PRG.sub_slowscrew2
    Rectangle (0,400 340x15), "-2-"
END_VISUALIZATION

// Device/Application/vis/cement_0
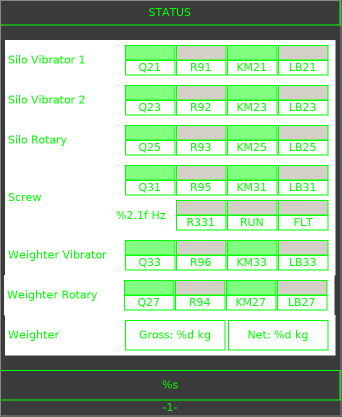
VISUALIZATION cement_0  // 342x417
    Rectangle (0,0 340x25), "STATUS"
    Rectangle (0,400 340x15), "-1-"
    Rectangle (0,370 340x30), "%s", text variable: Cement_PRG.cement_alarm
    RoundedRectangle (5,40 330x40), "Silo Vibrator 1"
    RoundedRectangle (125,45 50x15), colour toggle: DI121
    RoundedRectangle (125,60 50x15), "Q21"
    RoundedRectangle (176,45 50x15), colour toggle: DO311
    RoundedRectangle (176,60 50x15), "R91"
    RoundedRectangle (227,45 50x15), colour toggle: DI141
    RoundedRectangle (227,60 50x15), "KM21"
    RoundedRectangle (278,45 50x15), colour toggle: DI181
    RoundedRectangle (278,60 50x15), "LB21"
    RoundedRectangle (5,80 330x40), "Silo Vibrator 2"
    RoundedRectangle (125,85 50x15), colour toggle: DI122
    RoundedRectangle (125,100 50x15), "Q23"
    RoundedRectangle (176,85 50x15), colour toggle: DO312
    RoundedRectangle (176,100 50x15), "R92"
    RoundedRectangle (227,85 50x15), colour toggle: DI142
    RoundedRectangle (227,100 50x15), "KM23"
    RoundedRectangle (278,85 50x15), colour toggle: DI182
    RoundedRectangle (278,100 50x15), "LB23"
    RoundedRectangle (5,120 330x40), "Silo Rotary"
    RoundedRectangle (125,125 50x15), colour toggle: DI123
    RoundedRectangle (125,140 50x15), "Q25"
    RoundedRectangle (176,125 50x15), colour toggle: DO313
    RoundedRectangle (176,140 50x15), "R93"
    RoundedRectangle (227,125 50x15), colour toggle: DI143
    RoundedRectangle (227,140 50x15), "KM25"
    RoundedRectangle (278,125 50x15), colour toggle: DI183
    RoundedRectangle (278,140 50x15), "LB25"
    RoundedRectangle (5,160 330x75), "Screw"
    RoundedRectangle (125,165 50x15), colour toggle: DI125
    RoundedRectangle (125,180 50x15), "Q31"
    RoundedRectangle (176,165 50x15), colour toggle: DO315
    RoundedRectangle (176,180 50x15), "R95"
    RoundedRectangle (227,165 50x15), colour toggle: DI145
    RoundedRectangle (227,180 50x15), "KM31"
    RoundedRectangle (278,165 50x15), colour toggle: DI185
    RoundedRectangle (278,180 50x15), "LB31"
    RoundedRectangle (176,200 50x15), colour toggle: DO331
    RoundedRectangle (176,215 50x15), "R331"
    RoundedRectangle (227,200 50x15), colour toggle: DI161
    RoundedRectangle (227,215 50x15), "RUN"
    RoundedRectangle (278,200 50x15), colour toggle: DI162
    RoundedRectangle (278,215 50x15), "FLT"
    Rectangle (106,203 70x25), "%2.1f Hz", text variable: Cement_PRG.screw_Hz
    RoundedRectangle (5,235 330x40), "Weighter Vibrator"
    RoundedRectangle (125,240 50x15), colour toggle: DI126
    RoundedRectangle (125,255 50x15), "Q33"
    RoundedRectangle (176,240 50x15), colour toggle: DO316
    RoundedRectangle (176,255 50x15), "R96"
    RoundedRectangle (227,240 50x15), colour toggle: DI146
    RoundedRectangle (227,255 50x15), "KM33"
    RoundedRectangle (278,240 50x15), colour toggle: DI186
    RoundedRectangle (278,255 50x15), "LB33"
    RoundedRectangle (4,275 330x40), "Weighter Rotary"
    RoundedRectangle (124,280 50x15), colour toggle: DI124
    RoundedRectangle (124,295 50x15), "Q27"
    RoundedRectangle (175,280 50x15), colour toggle: DO314
    RoundedRectangle (175,295 50x15), "R94"
    RoundedRectangle (226,280 50x15), colour toggle: DI144
    RoundedRectangle (226,295 50x15), "KM27"
    RoundedRectangle (277,280 50x15), colour toggle: DI184
    RoundedRectangle (277,295 50x15), "LB27"
    RoundedRectangle (5,315 330x40), "Weighter"
    Rectangle (125,320 100x30), "Gross: %d kg", text variable: cem6
    Rectangle (228,320 100x30), "Net: %d kg", text variable: cem4
END_VISUALIZATION

// Device/Application/vis/cement_2
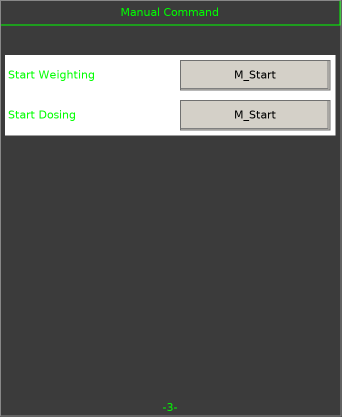
VISUALIZATION cement_2  // 342x417
    Rectangle (0,0 340x25), "Manual Command"
    Rectangle (0,400 340x15), "-3-"
    RoundedRectangle (5,55 330x40), "Start Weighting"
    RoundedRectangle (5,95 330x40), "Start Dosing"
    Button (180,60 150x30), "M_Start"
        tap Cement_PRG.manual_weighting
    Button (180,100 150x30), "M_Start"
        tap Cement_PRG.manual_dosing
END_VISUALIZATION

// Device/Application/vis/lime_0
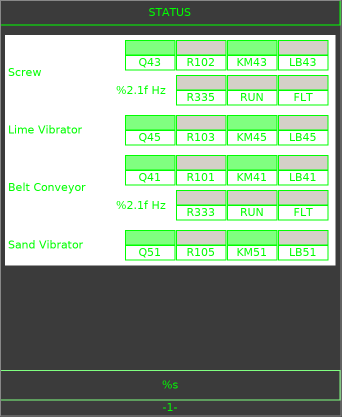
VISUALIZATION lime_0  // 342x417
    Rectangle (0,0 340x25), "STATUS"
    Rectangle (0,400 340x15), "-1-"
    Rectangle (0,370 340x30), "%s", text variable: LimeSand.lime_alarm
    RoundedRectangle (5,110 330x40), "Lime Vibrator"
    RoundedRectangle (125,115 50x15), colour toggle: DI133
    RoundedRectangle (125,130 50x15), "Q45"
    RoundedRectangle (176,115 50x15), colour toggle: DO323
    RoundedRectangle (176,130 50x15), "R103"
    RoundedRectangle (227,115 50x15), colour toggle: DI153
    RoundedRectangle (227,130 50x15), "KM45"
    RoundedRectangle (278,115 50x15), colour toggle: DI193
    RoundedRectangle (278,130 50x15), "LB45"
    RoundedRectangle (5,35 330x75), "Screw"
    RoundedRectangle (125,40 50x15), colour toggle: DI132
    RoundedRectangle (125,55 50x15), "Q43"
    RoundedRectangle (176,40 50x15), colour toggle: DO322
    RoundedRectangle (176,55 50x15), "R102"
    RoundedRectangle (227,40 50x15), colour toggle: DI152
    RoundedRectangle (227,55 50x15), "KM43"
    RoundedRectangle (278,40 50x15), colour toggle: DI192
    RoundedRectangle (278,55 50x15), "LB43"
    RoundedRectangle (176,75 50x15), colour toggle: DO335
    RoundedRectangle (176,90 50x15), "R335"
    RoundedRectangle (227,75 50x15), colour toggle: DI165
    RoundedRectangle (227,90 50x15), "RUN"
    RoundedRectangle (278,75 50x15), colour toggle: DI166
    RoundedRectangle (278,90 50x15), "FLT"
    Rectangle (106,78 70x25), "%2.1f Hz", text variable: LimeSand.screw_Hz
    RoundedRectangle (5,225 330x40), "Sand Vibrator"
    RoundedRectangle (125,230 50x15), colour toggle: DI135
    RoundedRectangle (125,245 50x15), "Q51"
    RoundedRectangle (176,230 50x15), colour toggle: DO325
    RoundedRectangle (176,245 50x15), "R105"
    RoundedRectangle (227,230 50x15), colour toggle: DI155
    RoundedRectangle (227,245 50x15), "KM51"
    RoundedRectangle (278,230 50x15), colour toggle: DI195
    RoundedRectangle (278,245 50x15), "LB51"
    RoundedRectangle (5,150 330x75), "Belt Conveyor"
    RoundedRectangle (125,155 50x15), colour toggle: DI131
    RoundedRectangle (125,170 50x15), "Q41"
    RoundedRectangle (176,155 50x15), colour toggle: DO321
    RoundedRectangle (176,170 50x15), "R101"
    RoundedRectangle (227,155 50x15), colour toggle: DI151
    RoundedRectangle (227,170 50x15), "KM41"
    RoundedRectangle (278,155 50x15), colour toggle: DI191
    RoundedRectangle (278,170 50x15), "LB41"
    RoundedRectangle (176,190 50x15), colour toggle: DO333
    RoundedRectangle (176,205 50x15), "R333"
    RoundedRectangle (227,190 50x15), colour toggle: DI163
    RoundedRectangle (227,205 50x15), "RUN"
    RoundedRectangle (278,190 50x15), colour toggle: DI164
    RoundedRectangle (278,205 50x15), "FLT"
    Rectangle (106,193 70x25), "%2.1f Hz", text variable: LimeSand.belt_Hz
END_VISUALIZATION

// Device/Application/vis/lime_1
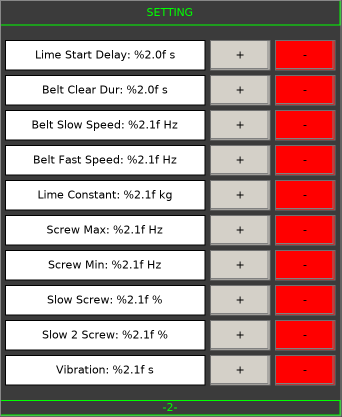
VISUALIZATION lime_1  // 342x417
    Rectangle (0,0 340x25), "SETTING"
    RoundedRectangle (5,40 200x30), "Lime Start Delay: %2.0f s", text variable: LimeSand.limedelay
    Button (210,40 60x30), "+"
        tap LimeSand.add_limedelay
    Button (275,40 60x30), "-"
        tap LimeSand.sub_limedelay
    RoundedRectangle (5,145 200x30), "Belt Fast Speed: %2.1f Hz", text variable: LimeSand.cleanspeed
    Button (210,145 60x30), "+"
        tap LimeSand.add_cleanspeed
    Button (275,145 60x30), "-"
        tap LimeSand.sub_cleanspeed
    Rectangle (0,400 340x15), "-2-"
    RoundedRectangle (5,110 200x30), "Belt Slow Speed: %2.1f Hz", text variable: LimeSand.bufferspeed
    Button (210,110 60x30), "+"
        tap LimeSand.add_bufferspeed
    Button (275,110 60x30), "-"
        tap LimeSand.sub_bufferspeed
    RoundedRectangle (5,180 200x30), "Lime Constant: %2.1f kg", text variable: LimeSand.limeconstant
    Button (210,180 60x30), "+"
        tap LimeSand.add_limeconstant
    Button (275,180 60x30), "-"
        tap LimeSand.sub_limeconstant
    RoundedRectangle (5,215 200x30), "Screw Max: %2.1f Hz", text variable: LimeSand.maxscrew
    Button (210,215 60x30), "+"
        tap LimeSand.add_maxscrew
    Button (275,215 60x30), "-"
        tap LimeSand.sub_maxscrew
    RoundedRectangle (5,250 200x30), "Screw Min: %2.1f Hz", text variable: LimeSand.minscrew
    Button (210,250 60x30), "+"
        tap LimeSand.add_minscrew
    Button (275,250 60x30), "-"
        tap LimeSand.sub_minscrew
    RoundedRectangle (5,285 200x30), "Slow Screw: %2.1f %", text variable: LimeSand.slowscrew
    Button (210,285 60x30), "+"
        tap LimeSand.add_slowscrew
    Button (275,285 60x30), "-"
        tap LimeSand.sub_slowscrew
    RoundedRectangle (5,320 200x30), "Slow 2 Screw: %2.1f %", text variable: LimeSand.slow2screw
    Button (210,320 60x30), "+"
        tap LimeSand.add_slow2screw
    Button (275,320 60x30), "-"
        tap LimeSand.sub_slow2screw
    RoundedRectangle (5,355 200x30), "Vibration: %2.1f s", text variable: LimeSand.vibreal
    Button (210,355 60x30), "+"
        tap LimeSand.add_vibreal
    Button (275,355 60x30), "-"
        tap LimeSand.sub_vibreal
    RoundedRectangle (5,75 200x30), "Belt Clear Dur: %2.0f s", text variable: LimeSand.clear_param
    Button (210,75 60x30), "+"
        tap LimeSand.add_clear
    Button (275,75 60x30), "-"
        tap LimeSand.sub_clear
END_VISUALIZATION

// Device/Application/vis/lime_3
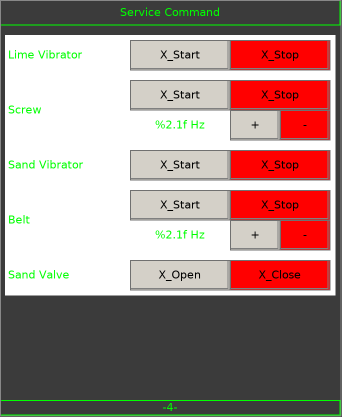
VISUALIZATION lime_3  // 342x417
    Rectangle (0,0 340x25), "Service Command"
    Rectangle (0,400 340x15), "-4-"
    RoundedRectangle (5,35 330x40), "Lime Vibrator"
    RoundedRectangle (5,75 330x70), "Screw"
    Rectangle (130,110 100x30), "%2.1f Hz", text variable: LimeSand.screw_service
    Button (130,40 100x30), "X_Start", colour toggle: DO323
        tap LimeSand.x_run_viblime
    Button (130,80 100x30), "X_Start", colour toggle: DO335
        tap LimeSand.x_run_screw
    Button (230,110 50x30), "+"
        tap LimeSand.add_screwservice
    Button (280,110 50x30), "-"
        tap LimeSand.sub_screwservice
    Button (230,40 100x30), "X_Stop"
        tap LimeSand.x_stop_viblime
    Button (230,80 100x30), "X_Stop"
        tap LimeSand.x_stop_screw
    RoundedRectangle (5,145 330x40), "Sand Vibrator"
    RoundedRectangle (5,185 330x70), "Belt"
    Rectangle (130,220 100x30), "%2.1f Hz", text variable: LimeSand.belt_Hz
    Button (130,150 100x30), "X_Start", colour toggle: DO325
        tap LimeSand.x_run_vibsand
    Button (130,190 100x30), "X_Start", colour toggle: DO333
        tap LimeSand.x_run_belt
    Button (230,220 50x30), "+"
        tap LimeSand.add_beltservice
    Button (280,220 50x30), "-"
        tap LimeSand.sub_beltservice
    Button (230,150 100x30), "X_Stop"
        tap LimeSand.x_stop_vibsand
    Button (230,190 100x30), "X_Stop"
        tap LimeSand.x_stop_belt
    RoundedRectangle (5,255 330x40), "Sand Valve"
    Button (130,260 100x30), "X_Open", colour toggle: DO326
        tap LimeSand.x_open_valve
    Button (230,260 100x30), "X_Close"
        tap LimeSand.x_close_valve
END_VISUALIZATION

// Device/Application/vis/lime_2
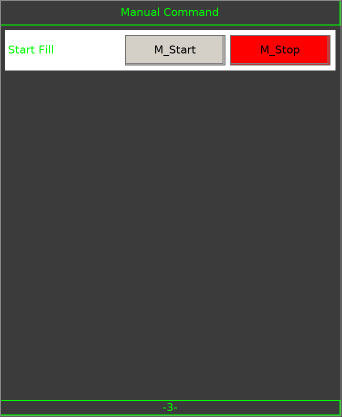
VISUALIZATION lime_2  // 342x417
    Rectangle (0,400 340x15), "-3-"
    Rectangle (0,0 340x25), "Manual Command"
    RoundedRectangle (5,30 330x40), "Start Fill"
    Button (125,35 100x30), "M_Start", colour toggle: LimeSand.manual_liming
        tap LimeSand.m_lime_start
    Button (230,35 100x30), "M_Stop"
        tap LimeSand.m_lime_stop
END_VISUALIZATION

// Device/Application/vis/cement_3
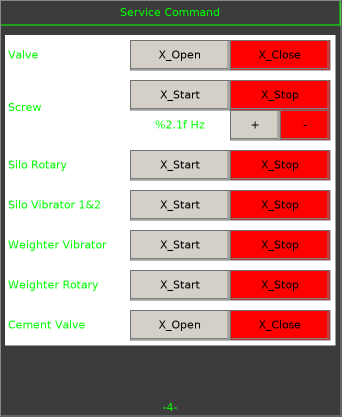
VISUALIZATION cement_3  // 342x417
    Rectangle (0,0 340x25), "Service Command"
    Rectangle (0,400 340x15), "-4-"
    RoundedRectangle (5,185 330x40), "Silo Vibrator 1&2"
    RoundedRectangle (5,145 330x40), "Silo Rotary"
    RoundedRectangle (5,70 330x75), "Screw"
    Rectangle (130,110 100x30), "%2.1f Hz", text variable: Cement_PRG.service_screw_Hz
    RoundedRectangle (5,225 330x40), "Weighter Vibrator"
    RoundedRectangle (5,265 330x40), "Weighter Rotary"
    Button (130,190 100x30), "X_Start", colour toggle: DO311
        tap Cement_PRG.x_run_vib
    Button (130,150 100x30), "X_Start", colour toggle: DO313
        tap Cement_PRG.x_run_rot
    Button (130,80 100x30), "X_Start", colour toggle: DO331
        tap Cement_PRG.x_run_screw
    Button (130,230 100x30), "X_Start", colour toggle: DO316
        tap Cement_PRG.x_run_vibweight
    Button (130,270 100x30), "X_Start", colour toggle: DO314
        tap Cement_PRG.x_run_rotweight
    Button (230,110 50x30), "+"
        tap Cement_PRG.add_serviceHz
    Button (280,110 50x30), "-"
        tap Cement_PRG.sub_serviceHz
    RoundedRectangle (5,35 330x40), "Valve"
    Button (130,40 100x30), "X_Open", colour toggle: DO371
        tap Cement_PRG.x_open_valve
    Button (230,40 100x30), "X_Close"
        tap Cement_PRG.x_close_valve
    Button (230,80 100x30), "X_Stop"
        tap Cement_PRG.x_stop_screw
    Button (230,150 100x30), "X_Stop"
        tap Cement_PRG.x_stop_rot
    Button (230,190 100x30), "X_Stop"
        tap Cement_PRG.x_stop_vib
    Button (230,230 100x30), "X_Stop"
        tap Cement_PRG.x_stop_vibweight
    Button (230,270 100x30), "X_Stop"
        tap Cement_PRG.x_stop_rotweight
    RoundedRectangle (5,305 330x40), "Cement Valve"
    Button (130,310 100x30), "X_Open", colour toggle: DO371
        tap Cement_PRG.x_open_valve
    Button (230,310 100x30), "X_Close"
        tap Cement_PRG.x_close_valve
END_VISUALIZATION

// Device/Application/vis/mixer_0
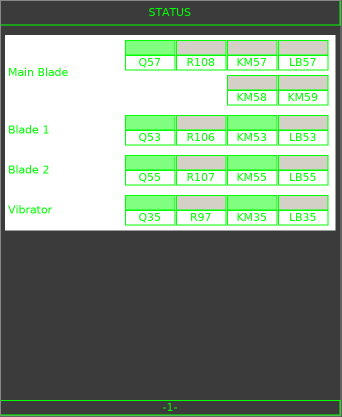
VISUALIZATION mixer_0  // 342x417
    Rectangle (0,0 340x25), "STATUS"
    Rectangle (0,400 340x15), "-1-"
    RoundedRectangle (5,35 330x75), "Main Blade"
    RoundedRectangle (5,110 330x40), "Blade 1"
    RoundedRectangle (125,115 50x15), colour toggle: DI171
    RoundedRectangle (125,130 50x15), "Q53"
    RoundedRectangle (176,115 50x15), colour toggle: DO345
    RoundedRectangle (176,130 50x15), "R106"
    RoundedRectangle (227,115 50x15), colour toggle: DI257
    RoundedRectangle (227,130 50x15), "KM53"
    RoundedRectangle (278,115 50x15), colour toggle: DI207
    RoundedRectangle (278,130 50x15), "LB53"
    RoundedRectangle (125,40 50x15), colour toggle: DI173
    RoundedRectangle (125,55 50x15), "Q57"
    RoundedRectangle (176,40 50x15), colour toggle: DO347
    RoundedRectangle (176,55 50x15), "R108"
    RoundedRectangle (227,40 50x15), colour toggle: DI254
    RoundedRectangle (227,55 50x15), "KM57"
    RoundedRectangle (278,40 50x15), colour toggle: DI238
    RoundedRectangle (278,55 50x15), "LB57"
    RoundedRectangle (227,90 50x15), "KM58"
    RoundedRectangle (278,90 50x15), "KM59"
    RoundedRectangle (227,75 50x15), colour toggle: DI256
    RoundedRectangle (278,75 50x15), colour toggle: DI255
    RoundedRectangle (5,150 330x40), "Blade 2"
    RoundedRectangle (125,155 50x15), colour toggle: DI172
    RoundedRectangle (125,170 50x15), "Q55"
    RoundedRectangle (176,155 50x15), colour toggle: DO346
    RoundedRectangle (176,170 50x15), "R107"
    RoundedRectangle (227,155 50x15), colour toggle: DI258
    RoundedRectangle (227,170 50x15), "KM55"
    RoundedRectangle (278,155 50x15), colour toggle: DI208
    RoundedRectangle (278,170 50x15), "LB55"
    RoundedRectangle (5,190 330x40), "Vibrator"
    RoundedRectangle (125,195 50x15), colour toggle: DI127
    RoundedRectangle (125,210 50x15), "Q35"
    RoundedRectangle (176,195 50x15), colour toggle: DO317
    RoundedRectangle (176,210 50x15), "R97"
    RoundedRectangle (227,195 50x15), colour toggle: DI147
    RoundedRectangle (227,210 50x15), "KM35"
    RoundedRectangle (278,195 50x15), colour toggle: DI187
    RoundedRectangle (278,210 50x15), "LB35"
END_VISUALIZATION

// Device/Application/vis/mixer_1
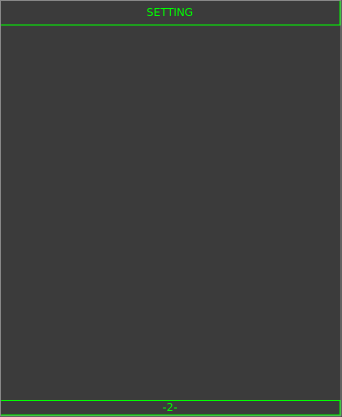
VISUALIZATION mixer_1  // 342x417
    Rectangle (0,0 340x25), "SETTING"
    Rectangle (0,400 340x15), "-2-"
END_VISUALIZATION

// Device/Application/vis/mixer_2
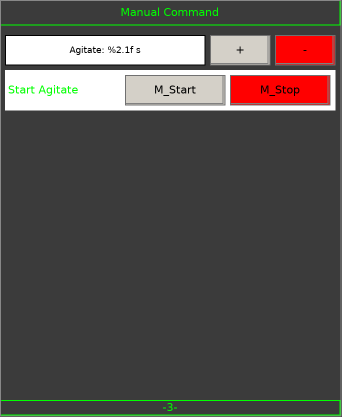
VISUALIZATION mixer_2  // 342x417
    Rectangle (0,0 340x25), "Manual Command"
    Rectangle (0,400 340x15), "-3-"
    RoundedRectangle (5,70 330x40), "Start Agitate"
    Button (125,75 100x30), "M_Start", colour toggle: Mixer_PRG.run_agitator
        tap Mixer_PRG.manual_run_agitator
    RoundedRectangle (5,35 200x30), "Agitate: %2.1f s", text variable: Mixer_PRG.agitatedura
    Button (210,35 60x30), "+"
        tap Mixer_PRG.add_agitatedura
    Button (275,35 60x30), "-"
        tap Mixer_PRG.sub_agitatedura
    Button (230,75 100x30), "M_Stop"
        tap Mixer_PRG.manual_stop_agitator
END_VISUALIZATION

// Device/Application/vis/mixer_3
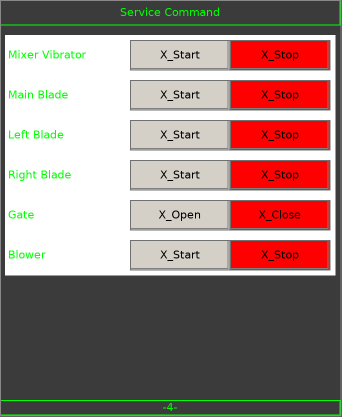
VISUALIZATION mixer_3  // 342x417
    Rectangle (0,0 340x25), "Service Command"
    Rectangle (0,400 340x15), "-4-"
    RoundedRectangle (5,35 330x40), "Mixer Vibrator"
    RoundedRectangle (5,195 330x40), "Gate"
    RoundedRectangle (5,75 330x40), "Main Blade"
    Button (130,80 100x30), "X_Start", colour toggle: DO347
        tap Mixer_PRG.x_run_mainagi
    Button (230,80 100x30), "X_Stop"
        tap Mixer_PRG.x_stop_mainagi
    RoundedRectangle (5,115 330x40), "Left Blade"
    Button (130,120 100x30), "X_Start", colour toggle: DO345
        tap Mixer_PRG.x_run_agi1
    Button (230,120 100x30), "X_Stop"
        tap Mixer_PRG.x_stop_agi1
    RoundedRectangle (5,155 330x40), "Right Blade"
    Button (130,160 100x30), "X_Start", colour toggle: DO346
        tap Mixer_PRG.x_run_agi2
    Button (230,160 100x30), "X_Stop"
        tap Mixer_PRG.x_stop_agi2
    Button (130,200 100x30), "X_Open", colour toggle: DO381
        tap Mixer_PRG.x_open_door
    Button (230,200 100x30), "X_Close"
        tap Mixer_PRG.x_close_door
    RoundedRectangle (5,235 330x40), "Blower"
    Button (130,240 100x30), "X_Start", colour toggle: DO382
        tap Mixer_PRG.x_start_blow
    Button (230,240 100x30), "X_Stop"
        tap Mixer_PRG.x_stop_blow
    Button (130,40 100x30), "X_Start", colour toggle: DO317
        tap Mixer_PRG.x_run_vibmixer
    Button (230,40 100x30), "X_Stop"
        tap Mixer_PRG.x_stop_vibmixer
END_VISUALIZATION

// Device/Application/vis/packing_0
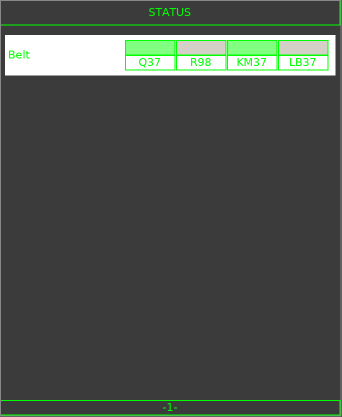
VISUALIZATION packing_0  // 342x417
    Rectangle (0,0 340x25), "STATUS"
    Rectangle (0,400 340x15), "-1-"
    RoundedRectangle (5,35 330x40), "Belt"
    RoundedRectangle (125,40 50x15), colour toggle: DI128
    RoundedRectangle (125,55 50x15), "Q37"
    RoundedRectangle (176,40 50x15), colour toggle: DO318
    RoundedRectangle (176,55 50x15), "R98"
    RoundedRectangle (227,40 50x15), colour toggle: DI148
    RoundedRectangle (227,55 50x15), "KM37"
    RoundedRectangle (278,40 50x15), colour toggle: DI188
    RoundedRectangle (278,55 50x15), "LB37"
END_VISUALIZATION

// Device/Application/vis/packing_3
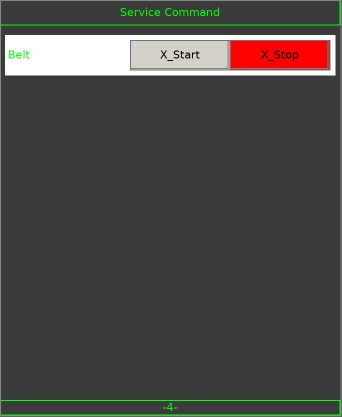
VISUALIZATION packing_3  // 342x417
    Rectangle (0,0 340x25), "Service Command"
    Rectangle (0,400 340x15), "-4-"
    RoundedRectangle (5,35 330x40), "Belt"
    Button (130,40 100x30), "X_Start", colour toggle: DO318
        tap Mixer_PRG.x_run_beltpacking
    Button (230,40 100x30), "X_Stop"
        tap Mixer_PRG.x_stop_beltpacking
END_VISUALIZATION

// Device/Application/vis/packing_2
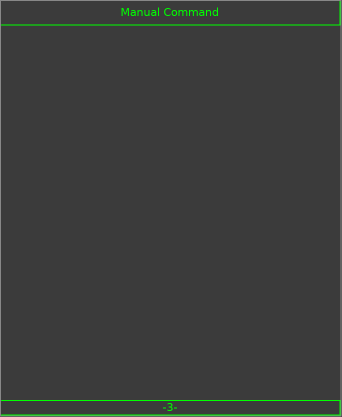
VISUALIZATION packing_2  // 342x417
    Rectangle (0,0 340x25), "Manual Command"
    Rectangle (0,400 340x15), "-3-"
END_VISUALIZATION

// Device/Application/vis/packing_1
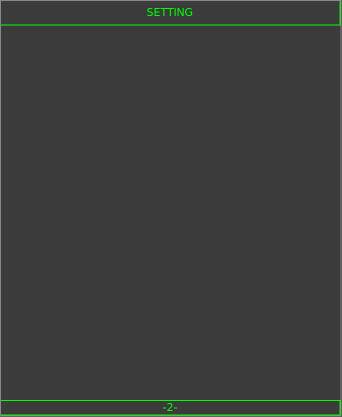
VISUALIZATION packing_1  // 342x417
    Rectangle (0,0 340x25), "SETTING"
    Rectangle (0,400 340x15), "-2-"
END_VISUALIZATION
